(*
    Function block for Power and Profile Monitor (PPM) controls under
    the LCLS_Tc_Motion (ND) framework:
    - Y in/powermeter/yag state mover via FB_PositionStatePMPSND
      with four states (OUT, POWERMETER, YAG1, YAG2)
    - power meter (FB_PPM_PowerMeter)
    - GigE camera power + illuminator (FB_PPM_Gige)
    - flow meter (FB_AnalogInput)
    - YAG thermocouple (FB_CC_TempSensor)
    - flow switch (FB_XTES_Flowswitch)

    FB_PPM is a thin wrapper for the state-mover plumbing and a tick
    site for the five orthogonal sub-devices. Motors, motion-stage
    interface array, position-state slot array, fast-fault output and
    arbiter are caller-owned; FB_PPM receives them by FB_Init
    REFERENCE TO and forwards them to fbStates via inline-init. The
    state enum bridge (eEnumSet / eEnumGet, UINT) and the four run-time
    toggles (bEnableMotion / bEnableBeamParams / bEnablePositionLimits
    / bReadDBNow, plain BOOL) are device-specific and live as classic
    VAR_INPUT; the body re-forwards them into fbStates each cycle.

    Per-state configuration is split across two configurators that
    co-operate on each ST_PositionState slot:
      - integrator's FB_CC_StatePMPSConfig array (per-install, declared
        in the caller PRG) wraps motion-lib's FB_StateSetup and writes
        fPosition + sPmpsState plus a caller-owned stDefault baseline
        (bMoveOk / bValid / bUseRawCounts / template fDelta).
      - FB_PPM.afbStateDefaults (device-side, hardcoded here) writes
        per-state sName and fDelta last, overriding the template
        baseline that FB_StateSetup just laid down. Ordering matters:
        the integrator must tick its PMPS array BEFORE calling fbPPM.
    Both configurators are idempotent once the parent state FB sets
    stPositionState.bUpdated := TRUE.

    Power meter and YAG thermocouple consume motion-stack state
    (eEnumGet, fbStates.stDbStateParams, axis NC state). The NC axis
    state DWORD is reached as `aiMotionStage[1].Axis.NcToPlc.AxisState`
    (I_MotionStage.Axis -> REFERENCE TO AXIS_REF).

    The following IO link points are included and should be used:
    - FB_PPM.fbPowerMeter.iVoltageINT -> power meter analog input voltage
    - FB_PPM.fbPowerMeter.fbThermoCouple.{bError,bUnderrange,bOverrange,iRaw}
      -> the corresponding thermocouple terminal inputs
    - FB_PPM.fbGige.iIlluminatorINT -> illuminator dimmer analog output voltage
    - FB_PPM.fbGige.bGigePower -> camera power digital output channel
    - FB_PPM.fbFlowMeter.iRaw -> flow meter current analog input channel
    - FB_PPM.fbYagTempSensor.{bError,bUnderrange,bOverrange,iRaw} -> YAG
      thermocouple terminal inputs
*)
{attribute 'call_after_init'}
FUNCTION_BLOCK FB_PPM
VAR_INPUT
    // Set this to a non-unknown value to request a new move.
    {attribute 'pytmc' := '
        pv: MMS:STATE:SET
        io: io
    '}
    eEnumSet : E_PPM_States;
    (* Flow meter offset in engineering units (per-install). *)
    fFlowOffset   : LREAL := 0;
    (* Power-meter responsivity (calibrated per gentec); if zero the
       responsive energy is not calculated. *)
    fResponsivity : LREAL;

    (* Passed straight through to FB_PPM_PowerMeter's analog input.
       Defaults are correct for EL3062; EL3602 needs iTermBits:=31
       with fTermMax/fTermMin matching the terminal's configured
       voltage range. *)
    iTermBits : UINT := 15;
    fTermMax  : REAL := 10000;
    fTermMin  : REAL := 0;

END_VAR
VAR
    {attribute 'pytmc' := 'pv: SPM'}
    fbPowerMeter : FB_PPM_PowerMeter;

    {attribute 'pytmc' := 'pv: CAM'}
    fbGige : FB_PPM_Gige;

    {attribute 'pytmc' := 'pv: FWM'}
    fbFlowMeter : FB_AnalogInput := (iTermBits := 15, fTermMax := 60, fTermMin := 0);

    {attribute 'pytmc' := 'pv: YAG:STC'}
    fbYagTempSensor : FB_CC_TempSensor;

    {attribute 'pytmc' := 'pv: FSW'}
    fbFlowSwitch : FB_XTES_Flowswitch;

    (* REFERENCE TO backing fields populated by FB_Init. Same names as
       FB_Init params; THIS^. disambiguates inside FB_Init.
       Live-bound to caller storage for the lifetime of the FB. *)
    {attribute 'no_copy'}
    aiMotionStage         : REFERENCE TO ARRAY[1..MotionConstants.MAX_STATE_MOTORS] OF I_MotionStage;
    {attribute 'no_copy'}
    astPositionState      : REFERENCE TO ARRAY[1..MotionConstants.MAX_STATE_MOTORS]
                                            OF ARRAY[1..GeneralConstants.MAX_STATES] OF ST_PositionState;
    {attribute 'no_copy'}
    fbFFHWO               : REFERENCE TO FB_HardwareFFOutput;
    {attribute 'no_copy'}
    fbArbiter             : REFERENCE TO FB_Arbiter;
    sDeviceName           : STRING;
    sTransitionKey        : STRING;
    bEnableMotion         : BOOL := TRUE;
    bEnableBeamParams     : BOOL;
    bEnablePositionLimits : BOOL;
    bReadDBNow            : BOOL;

    bFileReaderBusy       : REFERENCE TO BOOL;
    bFileReaderError      : REFERENCE TO BOOL;

    (* One configurator per PPM state. Writes the per-state sName and
       fDelta. Ticked cyclically in the body AFTER fbStates so its
       writes win over the template baseline FB_StateSetup applied via
       FB_CC_StatePMPSConfig. Idempotent once stPositionState.bUpdated
       trips. *)
    afbStateDefaults : ARRAY[1..4] OF FB_CC_DeviceStateDefaults[
        (stPositionState := astPositionState[1][E_PPM_States.OUT],
         sName           := 'OUT',
         fDelta          := FDELTA_DEFAULT),
        (stPositionState := astPositionState[1][E_PPM_States.POWERMETER],
         sName           := 'POWERMETER',
         fDelta          := FDELTA_DEFAULT),
        (stPositionState := astPositionState[1][E_PPM_States.YAG1],
         sName           := 'YAG1',
         fDelta          := FDELTA_DEFAULT),
        (stPositionState := astPositionState[1][E_PPM_States.YAG2],
         sName           := 'YAG2',
         fDelta          := FDELTA_DEFAULT)
    ];

    {attribute 'pytmc' := 'pv: MMS'}
    fbStates : FB_PositionStatePMPSND(
        aiMotionStage         := aiMotionStage,
        astPositionState      := astPositionState,
        nActiveMotorCount     := 1,
        eEnumSet              := eEnumSet,
        eEnumGet              := eEnumGet,
        bEnableMotion         := bEnableMotion,
        eMotionRequestPolicy  := E_MotionRequestPolicy.INTERRUPT,
        bEnableBeamParams     := bEnableBeamParams,
        bEnablePositionLimits := bEnablePositionLimits,
        bReadDBNow            := bReadDBNow,
        bFileReaderBusy       := bFileReaderBusy,
        bFileReaderError      := bFileReaderError,
        fbFFHWO               := fbFFHWO,
        fbArbiter             := fbArbiter,
        sDeviceName           := sDeviceName,
        sTransitionKey        := sTransitionKey
    );

    i : UINT;
END_VAR

VAR_OUTPUT
    // The current position state as an enum.
    {attribute 'pytmc' := '
        pv: MMS:STATE:GET
        io: i
    '}
    eEnumGet: E_PPM_States;
    // The PMPS database lookup associated with the current position state.
    stDbStateParams: ST_DbStateParams;
END_VAR

VAR CONSTANT
    (* PPM-wide default tolerance for state in-position detection,
       applied per-state by afbStateDefaults. *)
    FDELTA_DEFAULT : LREAL := 2;
END_VAR

(* Nil-ref guards: every REFERENCE TO backing field must be bound. *)
IF NOT __ISVALIDREF(aiMotionStage)
   OR NOT __ISVALIDREF(astPositionState)
   OR NOT __ISVALIDREF(fbFFHWO)
   OR NOT __ISVALIDREF(fbArbiter) THEN
    RETURN;
END_IF

(* Device-side per-state defaults (afbStateDefaults) are written
   once in FB_CC_DeviceStateDefaults.CallAfterInit; no cyclic tick. *)
fbStates(stDbStateParams=> stDbStateParams);

(* Power meter: consumes the current state enum + axis NC state for
   background auto-collection, and the PMPS DB temp setpoint to drive
   its thermocouple FFO. Vetoes the temp FFO outside POWERMETER. *)
fbPowerMeter(
    fTempSP       := fbStates.stDbStateParams.stReactiveParams.nTempSP,
    bVetoTempFFO  := eEnumGet <> E_PPM_States.POWERMETER,
    sDeviceName   := sDeviceName,
    fbFFHWO       := fbFFHWO,
    eEnumGet      := eEnumGet,
    stYAxisState  := aiMotionStage[1].Axis.NcToPlc.AxisState,
    fResponsivity := fResponsivity,
    iTermBits     := iTermBits,
    fTermMax      := fTermMax,
    fTermMin      := fTermMin
);

fbGige();
fbFlowMeter(fOffset := fFlowOffset);

(* YAG thermocouple: only faults when the YAG is actually in-beam
   (i.e. not OUT). Driven by the same PMPS DB temp setpoint. *)
fbYagTempSensor(
    fFaultThreshold := fbStates.stDbStateParams.stReactiveParams.nTempSP,
    bVeto           := eEnumGet = E_PPM_States.OUT,
    sDevName        := sDeviceName,
    io_fbFFHWO      := fbFFHWO
);

fbFlowSwitch();

(*
    {attribute 'call_after_init'} on FB_PPM causes TwinCAT to auto-fire
    THIS^.CallAfterInit() after FB_PPM.FB_Init completes.

    fbStates was constructed via inline-init in FB_PPM's VAR section,
    which ran BEFORE FB_PPM.FB_Init bound the REF fields on THIS^.
    Consequently fbStates' inline-init forwarded nil REFs into
    fbStates.FB_Init, and the auto-fired fbStates.CallAfterInit guards
    on those nil REFs and bails. This method re-supplies the now-valid
    refs through fbStates.CallAfterInitStateMover, which re-binds them and runs
    the full child-FB wiring chain (Core / ND / PMPSND).
*)
{attribute 'call_after_init'}
METHOD CallAfterInit
afbStateDefaults[1].CallAfterInit(stPositionState := THIS^.astPositionState[1][E_PPM_States.OUT]);
afbStateDefaults[2].CallAfterInit(stPositionState := THIS^.astPositionState[1][E_PPM_States.POWERMETER]);
afbStateDefaults[3].CallAfterInit(stPositionState := THIS^.astPositionState[1][E_PPM_States.YAG1]);
afbStateDefaults[4].CallAfterInit(stPositionState := THIS^.astPositionState[1][E_PPM_States.YAG2]);

THIS^.fbStates.CallAfterInitStateMover(
    aiMotionStage         := aiMotionStage,
    astPositionState      := astPositionState,
    nActiveMotorCount     := 1,
    eEnumSet              := eEnumSet,
    eEnumGet              := eEnumGet,
    bEnableMotion         := bEnableMotion,
    eMotionRequestPolicy  := E_MotionRequestPolicy.INTERRUPT,
);

THIS^.fbStates.CallAfterInitPMPS(
    aiMotionStage         := aiMotionStage,
    astPositionState      := astPositionState,
    bEnableBeamParams     := bEnableBeamParams,
    bEnablePositionLimits := bEnablePositionLimits,
    bReadDBNow            := bReadDBNow,
    bFileReaderBusy       := bFileReaderBusy,
    bFileReaderError      := bFileReaderError,
    fbFFHWO               := fbFFHWO,
    fbArbiter             := fbArbiter,
    sDeviceName           := sDeviceName,
    sTransitionKey        := sTransitionKey
);
END_METHOD

(* Stores all FB_Init inputs into instance fields. Every non-value
   input is REFERENCE TO and is REF= bound for the lifetime of the FB
   (matches the rule: non-interface FB_Init inputs are taken by ref).
   Inline-init of fbStates above runs first, capturing the FB_Init
   params at construction time; this method then records the same
   references on THIS^ for body-side use and live caller writes.
   The file-reader busy/error inputs are bound straight to
   MOTION_GVL.fbPmpsFileReader inside fbStates' inline-init. *)
{attribute 'analysis' := '-33'}
METHOD FB_Init : BOOL
VAR_INPUT
    bInitRetains           : BOOL;
    bInCopyCode            : BOOL;
    aiMotionStage          : REFERENCE TO ARRAY[1..MotionConstants.MAX_STATE_MOTORS] OF I_MotionStage;
    astPositionState       : REFERENCE TO ARRAY[1..MotionConstants.MAX_STATE_MOTORS]
                                            OF ARRAY[1..GeneralConstants.MAX_STATES] OF ST_PositionState;
    fbFFHWO                : REFERENCE TO FB_HardwareFFOutput;
    fbArbiter              : REFERENCE TO FB_Arbiter;
    sDeviceName            : STRING;
    sTransitionKey         : STRING;
    bEnableBeamParams      : BOOL;
    bEnablePositionLimits  : BOOL;
    bReadDBNow             : BOOL;
    bFileReaderBusy       : REFERENCE TO BOOL;
    bFileReaderError      : REFERENCE TO BOOL;
END_VAR
THIS^.aiMotionStage    REF= aiMotionStage;
THIS^.astPositionState REF= astPositionState;
THIS^.fbFFHWO          REF= fbFFHWO;
THIS^.fbArbiter        REF= fbArbiter;
THIS^.sDeviceName      := sDeviceName;
THIS^.sTransitionKey   := sTransitionKey;
THIS^.bEnableBeamParams     := bEnableBeamParams;
THIS^.bEnablePositionLimits := bEnablePositionLimits;
THIS^.bReadDBNow            := bReadDBNow;
THIS^.bFileReaderBusy       REF= bFileReaderBusy;
THIS^.bFileReaderError      REF= bFileReaderError;
END_METHOD

END_FUNCTION_BLOCK

(* stored: Version 1.1.0.1
   POU FB_PPM: Id {21ba0056-420c-4281-af9c-7f35e47eaf5b}, SpecialFunc None
   Method CallAfterInit: Id {21ba0057-420c-4281-af9c-7f35e47eaf5c}
   Method FB_init: Id {21ba0058-420c-4281-af9c-7f35e47eaf5d} *)
